// TIA Portal V19 export
FUNCTION "Conv_NUM_to_STRING" : String   // FC58, LAD
// stored: Access Published, SetENOAutomatically false
   VAR_INPUT
      NumericValue : Variant;
      NDec : USInt;
   END_VAR
   VAR_TEMP
      retval_MOVE_BLK : Int;
      value_LREAL : LReal;
      value_REAL : Real;
      value_USINT : USInt;
      value_SINT : SInt;
      value_UINT : UInt;
      value_INT : Int;
      value_UDINT : UDInt;
      value_DINT : DInt;
   END_VAR
BEGIN

REGION Network 1 (SCL)
   #Conv_NUM_to_STRING := 'E';
END_REGION

REGION Network 2 (SCL): LREAL -> STRING
   IF TypeOf(#NumericValue) = TypeOf(#value_LREAL) THEN


       #retval_MOVE_BLK := MOVE_BLK_VARIANT(SRC := #NumericValue, COUNT := 1, SRC_INDEX := 0, DEST_INDEX := 0, DEST => #value_LREAL);

       IF #retval_MOVE_BLK <> 0 THEN
           RETURN;
       END_IF;


       VAL_STRG(IN := #value_LREAL,
                SIZE :=0,
                PREC := #NDec,
                FORMAT := 0,
                P := 1,
                OUT => #Conv_NUM_to_STRING);



       RETURN;


   END_IF;
END_REGION

REGION Network 3 (SCL): REAL -> STRING
   IF TypeOf(#NumericValue) = TypeOf(#value_REAL) THEN


       #retval_MOVE_BLK := MOVE_BLK_VARIANT(SRC := #NumericValue, COUNT := 1, SRC_INDEX := 0, DEST_INDEX := 0, DEST => #value_REAL);

       IF #retval_MOVE_BLK <> 0 THEN
           RETURN;
       END_IF;


       VAL_STRG(IN := #value_REAL,
                SIZE :=0,
                PREC := #NDec,
                FORMAT := 0,
                P := 1,
                OUT => #Conv_NUM_to_STRING);

       RETURN;


   END_IF;
END_REGION

REGION Network 4 (SCL): USINT -> STRING
   IF TypeOf(#NumericValue) = TypeOf(#value_USINT) THEN


       #retval_MOVE_BLK := MOVE_BLK_VARIANT(SRC := #NumericValue, COUNT := 1, SRC_INDEX := 0, DEST_INDEX := 0, DEST => #value_USINT);

       IF #retval_MOVE_BLK <> 0 THEN
           RETURN;
       END_IF;


       VAL_STRG(IN := #value_USINT,
                SIZE :=0,
                PREC := #NDec,
                FORMAT := 0,
                P := 1,
                OUT => #Conv_NUM_to_STRING);

       RETURN;


   END_IF;
END_REGION

REGION Network 5 (SCL): SINT -> STRING
   IF TypeOf(#NumericValue) = TypeOf(#value_SINT) THEN


       #retval_MOVE_BLK := MOVE_BLK_VARIANT(SRC := #NumericValue, COUNT := 1, SRC_INDEX := 0, DEST_INDEX := 0, DEST => #value_SINT);

       IF #retval_MOVE_BLK <> 0 THEN
           RETURN;
       END_IF;


       VAL_STRG(IN := #value_SINT,
                SIZE :=0,
                PREC := #NDec,
                FORMAT := 0,
                P := 1,
                OUT => #Conv_NUM_to_STRING);

       RETURN;


   END_IF;
END_REGION

REGION Network 6 (SCL): UINT -> STRING
   IF TypeOf(#NumericValue) = TypeOf(#value_UINT) THEN


       #retval_MOVE_BLK := MOVE_BLK_VARIANT(SRC := #NumericValue, COUNT := 1, SRC_INDEX := 0, DEST_INDEX := 0, DEST => #value_UINT);

       IF #retval_MOVE_BLK <> 0 THEN
           RETURN;
       END_IF;


       VAL_STRG(IN := #value_UINT,
                SIZE :=0,
                PREC := #NDec,
                FORMAT := 0,
                P := 1,
                OUT => #Conv_NUM_to_STRING);

       RETURN;


   END_IF;
END_REGION

REGION Network 7 (SCL): INT -> STRING
   IF TypeOf(#NumericValue) = TypeOf(#value_INT) THEN


       #retval_MOVE_BLK := MOVE_BLK_VARIANT(SRC := #NumericValue, COUNT := 1, SRC_INDEX := 0, DEST_INDEX := 0, DEST => #value_INT);

       IF #retval_MOVE_BLK <> 0 THEN
           RETURN;
       END_IF;


       VAL_STRG(IN := #value_INT,
                SIZE :=0,
                PREC := #NDec,
                FORMAT := 0,
                P := 1,
                OUT => #Conv_NUM_to_STRING);

       RETURN;


   END_IF;
END_REGION

REGION Network 8 (SCL): UDINT -> STRING
   IF TypeOf(#NumericValue) = TypeOf(#value_UDINT) THEN


       #retval_MOVE_BLK := MOVE_BLK_VARIANT(SRC := #NumericValue, COUNT := 1, SRC_INDEX := 0, DEST_INDEX := 0, DEST => #value_UDINT);

       IF #retval_MOVE_BLK <> 0 THEN
           RETURN;
       END_IF;


       VAL_STRG(IN := #value_UDINT,
                SIZE :=0,
                PREC := #NDec,
                FORMAT := 0,
                P := 1,
                OUT => #Conv_NUM_to_STRING);

       RETURN;


   END_IF;
END_REGION

REGION Network 9 (SCL): DINT -> STRING
   IF TypeOf(#NumericValue) = TypeOf(#value_DINT) THEN


       #retval_MOVE_BLK := MOVE_BLK_VARIANT(SRC := #NumericValue, COUNT := 1, SRC_INDEX := 0, DEST_INDEX := 0, DEST => #value_DINT);

       IF #retval_MOVE_BLK <> 0 THEN
           RETURN;
       END_IF;


       VAL_STRG(IN := #value_DINT,
                SIZE :=0,
                PREC := #NDec,
                FORMAT := 0,
                P := 1,
                OUT => #Conv_NUM_to_STRING);

       RETURN;


   END_IF;
END_REGION
END_FUNCTION
